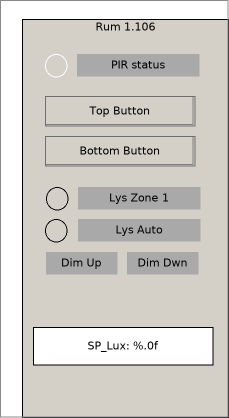
VISUALIZATION Visualization_1_317  // 229x418
    RoundedRectangle (22,19 207x399), "Rum 1.106"
    Rectangle (33,327 180x38), "SP_Lux: %.0f", text variable: P_Rum_1_317.fbLys.fbLightCtrl.fLuxZone1
    Button (45,96 150x30), "Top Button"
        tap P_Rum_1_317.bTopButtonZone1_Visu
    Button (45,136 150x30), "Bottom Button"
        tap P_Rum_1_317.bBottomButtonZone1_Visu
    Ellipse (46,187 22x23), colour toggle: P_Rum_1_317.fbLys.fbLightCtrl.bOnZone1
    Rectangle (78,187 122x22), "Lys Zone 1"
    Rectangle (46,252 71x22), "Dim Up", colour toggle: P_Rum_1_317.fbLys.fbLightCtrl.bDimUp
    Rectangle (127,252 71x22), "Dim Dwn", colour toggle: P_Rum_1_317.fbLys.fbLightCtrl.bDimDwn
    Ellipse (45,219 22x23), colour toggle: P_Rum_1_317.fbLys.fbLightCtrl.bAutoZone1
    Rectangle (78,219 122x22), "Lys Auto"
    Ellipse (45,54 22x23), colour toggle: P_Rum_1_317.fbLys.fbLightCtrl.bPIR
    Rectangle (77,54 122x22), "PIR status"
END_VISUALIZATION

(* stored: Version 1.1.0.1
   Visu Visualization_1_317: Id {88778d8b-3eb6-42f0-82cd-96a062d82408} *)
